# EPICS autosave request: tucsenApp/Db/tucsen_settings.req
$(P)$(R)BinMode
$(P)$(R)AutoExposure
$(P)$(R)HorizontalMirror
$(P)$(R)VerticalMirror
$(P)$(R)FanGear
$(P)$(R)AutoLevels
$(P)$(R)Histogram
$(P)$(R)Enhance
$(P)$(R)DefectCorrection
$(P)$(R)EnableDenoise
$(P)$(R)FlatCorrection
$(P)$(R)DataFormat
$(P)$(R)DynRgeCorrection
$(P)$(R)Brightness
$(P)$(R)BlackLevel
$(P)$(R)Sharpness
$(P)$(R)NoiseLevel
$(P)$(R)HDRK
$(P)$(R)Gamma
$(P)$(R)Contrast
$(P)$(R)LeftLevels
$(P)$(R)RightLevels
$(P)$(R)FrameFormat
file "ADBase_settings.req", P=$(P), R=$(R)
